// TIA Portal project "Motion_Control" (V17)

(* hardware
DEVICE "HMI_1"  KTP700 Basic PN
   slot 0: "HMI_1"  KTP700 Basic PN  6AV2 123-2GB03-0AX0  17.0.0.0
   slot 1: "HMI_RT_1"  KTP700 Basic PN  6AV2 123-2GB03-0AX0  17.0.0.0
   slot 5: "HMI_1.IE_CP_1"  PROFINET Interface  17.0.0.0
      slot 1: "PROFINET Interface_1"  PROFINET Interface
         slot 1: "Port_1"  Port
DEVICE "S7-1200 station_1"  S7-1200 Station
   slot 0: "Rack_0"  S7-1200 Rack  Rack  V1.0
   slot 1: "PLC_2"  CPU 1212C DC/DC/DC  6ES7 212-1AE40-0XB0  V4.5
*)

// ===== PLC "PLC_2"  CPU 1212C DC/DC/DC =====

VAR_GLOBAL   // PLC tag table "Default tag table"
   "Axis_1_Pulse" AT %Q0.0 : Bool;
   "Axis_1_Direction" AT %Q0.1 : Bool;
   "Axis_1_Homing switch" AT %I0.0 : Bool;
   "Axis_1_LowHwLimitSwitch" AT %I0.1 : Bool;
   "Axis_1_HighHwLimitSwitch" AT %I0.2 : Bool;
   "HMI Driver Start Stop" AT %M10.0 : Bool;
   "Axis 1 Driver Disable" AT %Q0.2 : Bool;
   "Error Power" AT %MW20 : Word;
   "HMI Home Position" AT %M10.1 : Bool;
   "Error Homing" AT %MW22 : Word;
   "HMI CCW" AT %M10.2 : Bool;
   "HMI CW" AT %M10.3 : Bool;
   "Error MoveJog" AT %MW24 : Word;
   "HMI Relative Button" AT %M10.4 : Bool;
   "Error Relative" AT %MW26 : Word;
   "HMI Distance Input" AT %MD28 : Real;
   "Real Distance Input" AT %MD32 : Real;
   "HMI Absolute Button" AT %M10.5 : Bool;
   "Error Absolute" AT %MW36 : Word;
   "HMI Stop Button" AT %M10.6 : Bool;
   "Error Halt" AT %MW38 : Word;
   "HMI System Reset" AT %M10.7 : Bool;
   "Error Reset" AT %MW40 : Word;
   "Position Memory" AT %MD42 : Real;
   "Position Value" AT %MD46 : Real;
   "Velocity Value" AT %MD50 : Real;
   "Velocity Go" AT %M11.0 : Bool;
   "HMI Movement 1" AT %M11.1 : Bool;
   "Tag_1" AT %M11.2 : Bool;
   "Error CT" AT %MW54 : Word;
END_VAR

// folder: System blocks/Program resources

DATA_BLOCK "Timer System Stop"   // DB9
{ S7_Optimized_Access := 'TRUE' }
AUTHOR : Simatic
FAMILY : IEC
NAME : IEC_TMR
VERSION : 1.0
// stored: InstanceOfName IEC_TIMER
"IEC_TIMER"
BEGIN
END_DATA_BLOCK

// folder: (top level)

DATA_BLOCK "Axis_1"   // DB1, Motion_DB
{ S7_Optimized_Access := 'TRUE' }
AUTHOR : SIMATIC
FAMILY : BasicMC
NAME : TO_PosAx
VERSION : 7.0
// stored: InstanceOfName TO_PositioningAxis
"TO_PositioningAxis"
BEGIN
   // Axis.PositionLimitsMax_AddressCU = %I0.2
   // Axis.PositionLimitsMin_AddressCU = %I0.1
   // Axis.PassiveHomingReferencePointSwitch_AddressCU = %I0.0
   // Axis.HomingReferencePointSwitch_AddressCU = %I0.0
   // Axis.NormalizedMaxVelocity.Input = 360.0
   // Axis.LengthUnitNormalized.Distance = 1005
   // Axis.OnlinePtoModeCU = 16#0000_0002
   // Axis.DirectionOutputEnabledCU = TRUE
   // Axis.SelectedChannel2EnumCU = %Q0.1
   // Axis.SelectedChannel1EnumCU = %Q0.0
   // Pulse.MinDeltaDeltaFrequencyCU = 0.004
   // Pulse.MaxDeltaDeltaFrequencyCU = 1.0E+10
   // Pulse.MinDeltaFrequencyCU = 0.005
   // Pulse.MaxDeltaFrequencyCU = 9.5E+9
   // Pulse.MinFrequencyCU = 1.0
   // Pulse.MaxFrequencyCU = 100000.0
   // Pulse.OutputSourceCU = 16#0000_0000
   // Axis.SelectPTO = 0
   // Axis.LengthUnit.LastDistance = 1005
END_DATA_BLOCK

DATA_BLOCK "Movement Table"   // DB10, BMC_202
{ S7_Optimized_Access := 'TRUE' }
AUTHOR : SIMATIC
FAMILY : BasicMC
NAME : CmdTab
VERSION : 7.0
// stored: InstanceOfName TO_CommandTable
"TO_CommandTable"
BEGIN
   // BasicMotionControl.CompileUnit.ExtendedGeneral.ConnectedAxisDBName = Axis_1
   // BasicMotionControl.CompileUnit.ExtendedGeneral.UsedParameters = 1
   // BasicMotionControl.CompileUnit.ExtendedGeneral.AxisID = {2232340-4704}
END_DATA_BLOCK

ORGANIZATION_BLOCK "Main"   // OB1, LAD, ProgramCycle
TITLE = "Main Program Sweep (Cycle)"
{ S7_Optimized_Access := 'TRUE' }
VERSION : 0.1
   VAR_INPUT
      Initial_Call : Bool;   // Initial call of this OB
      Remanence : Bool;   // =True, if remanent data are available
   END_VAR
   VAR_TEMP   // added for the SCL form of the ladder/FBD networks
      _w1 : Bool;
   END_VAR
BEGIN

REGION Network 1: Commissioning the driver
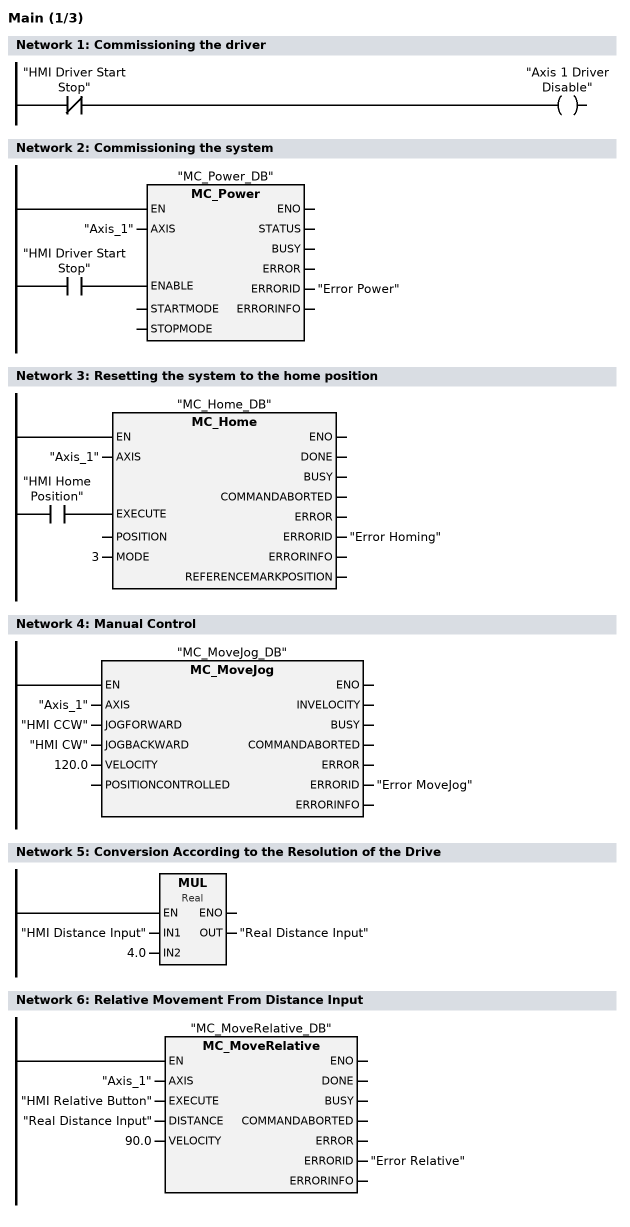
   RUNG wire#powerrail
      I_Contact( "HMI Driver Start Stop" )
      Coil( "Axis 1 Driver Disable" )
   END_RUNG
   // the same network as SCL:
   "Axis 1 Driver Disable" := NOT "HMI Driver Start Stop";
END_REGION

REGION Network 2: Commissioning the system
   "MC_Power_DB"(Axis := "Axis_1", Enable := "HMI Driver Start Stop", ErrorID => "Error Power");   // MC_Power
END_REGION

REGION Network 3: Resetting the system to the home position
   "MC_Home_DB"(Axis := "Axis_1", Execute := "HMI Home Position", Mode := 3, ErrorID => "Error Homing");   // MC_Home
END_REGION

REGION Network 4: Manual Control
   "MC_MoveJog_DB"(Axis := "Axis_1",   // MC_MoveJog
                   JogForward := "HMI CCW",
                   JogBackward := "HMI CW",
                   Velocity := 120.0,
                   ErrorID => "Error MoveJog");
END_REGION

REGION Network 5: Conversion According to the Resolution of the Drive
   RUNG wire#powerrail
      { S7_Templates := "SrcType := Real" } Mul(in1 := "HMI Distance Input", in2 := 4.0, out => "Real Distance Input")
   END_RUNG
   // the same network as SCL:
   "Real Distance Input" := "HMI Distance Input" * 4.0;
END_REGION

REGION Network 6: Relative Movement From Distance Input
   "MC_MoveRelative_DB"(Axis := "Axis_1",   // MC_MoveRelative
                        Execute := "HMI Relative Button",
                        Distance := "Real Distance Input",
                        Velocity := 90.0,
                        ErrorID => "Error Relative");
END_REGION

REGION Network 7: Absolute Movement From Distance Input
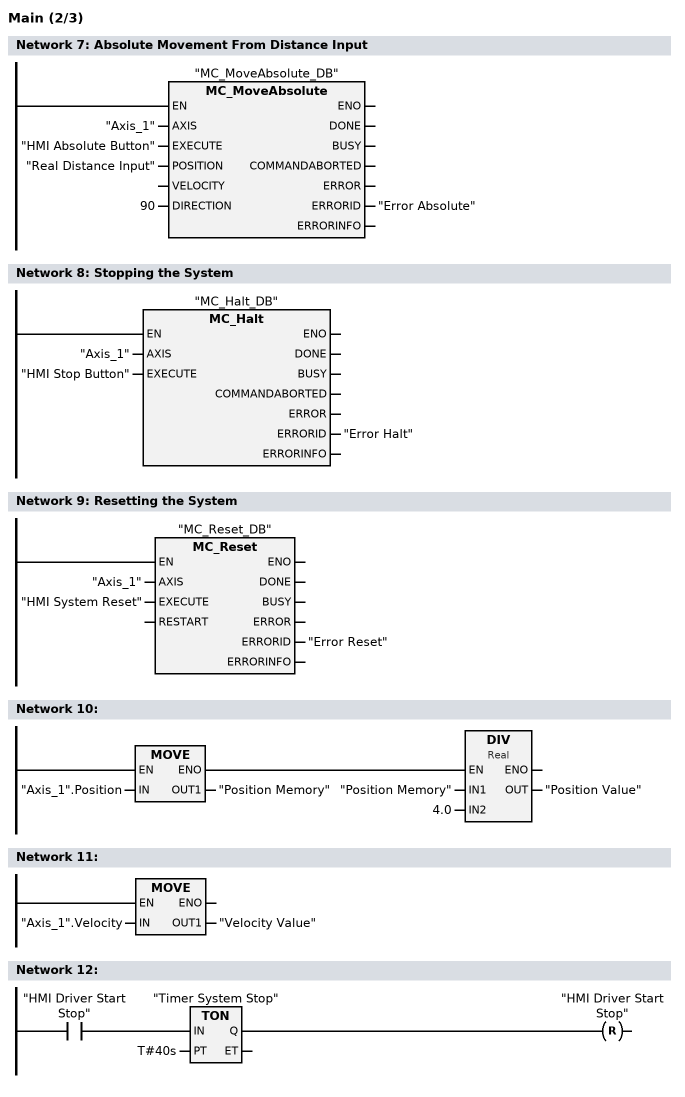
   "MC_MoveAbsolute_DB"(Axis := "Axis_1",   // MC_MoveAbsolute
                        Execute := "HMI Absolute Button",
                        Position := "Real Distance Input",
                        Direction := 90,
                        ErrorID => "Error Absolute");
END_REGION

REGION Network 8: Stopping the System
   "MC_Halt_DB"(Axis := "Axis_1", Execute := "HMI Stop Button", ErrorID => "Error Halt");   // MC_Halt
END_REGION

REGION Network 9: Resetting the System
   "MC_Reset_DB"(Axis := "Axis_1", Execute := "HMI System Reset", ErrorID => "Error Reset");   // MC_Reset
END_REGION

REGION Network 10
   RUNG wire#powerrail
      Move(in := "Axis_1".Position, out1 => "Position Memory")
      { S7_Templates := "SrcType := Real" } Div(in1 := "Position Memory", in2 := 4.0, out => "Position Value")
   END_RUNG
   // the same network as SCL:
   "Position Memory" := "Axis_1".Position;
   "Position Value" := "Position Memory" / 4.0;
END_REGION

REGION Network 11
   RUNG wire#powerrail
      Move(in := "Axis_1".Velocity, out1 => "Velocity Value")
   END_RUNG
   // the same network as SCL:
   "Velocity Value" := "Axis_1".Velocity;
END_REGION

REGION Network 12
   "Timer System Stop".TON(IN := "HMI Driver Start Stop", PT := T#40s);
   IF "Timer System Stop".Q THEN "HMI Driver Start Stop" := FALSE; END_IF;
END_REGION

REGION Network 13
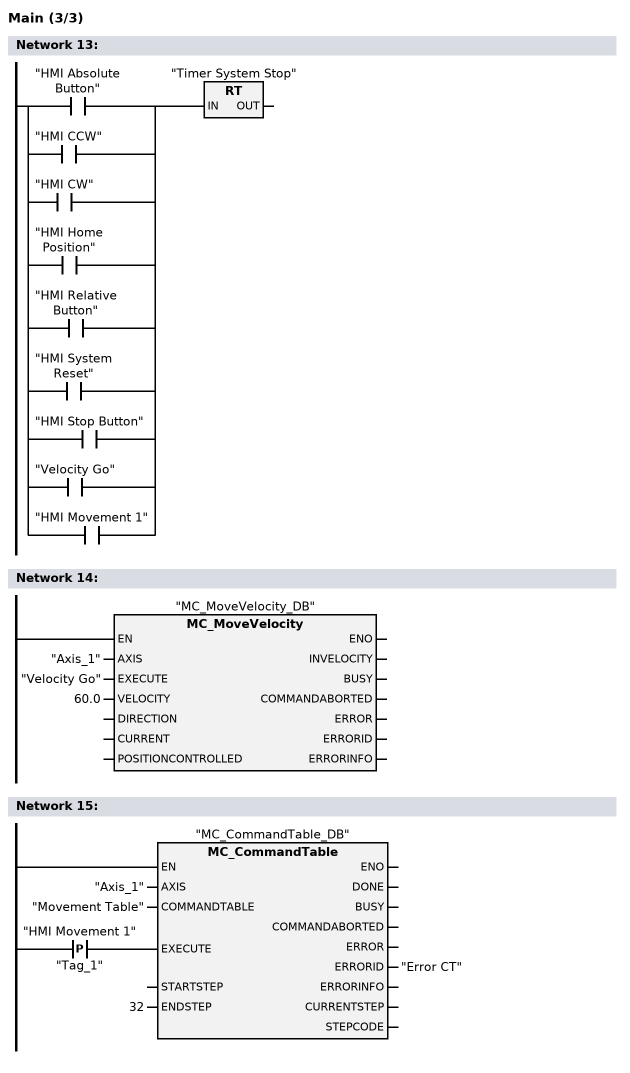
   RUNG wire#powerrail
      Contact( "HMI Absolute Button" )
      wire#w1
      RT_Coil( "Timer System Stop" )
   END_RUNG
   RUNG wire#powerrail
      Contact( "HMI CCW" )
   END_RUNG wire#w1
   RUNG wire#powerrail
      Contact( "HMI CW" )
   END_RUNG wire#w1
   RUNG wire#powerrail
      Contact( "HMI Home Position" )
   END_RUNG wire#w1
   RUNG wire#powerrail
      Contact( "HMI Relative Button" )
   END_RUNG wire#w1
   RUNG wire#powerrail
      Contact( "HMI System Reset" )
   END_RUNG wire#w1
   RUNG wire#powerrail
      Contact( "HMI Stop Button" )
   END_RUNG wire#w1
   RUNG wire#powerrail
      Contact( "Velocity Go" )
   END_RUNG wire#w1
   RUNG wire#powerrail
      Contact( "HMI Movement 1" )
   END_RUNG wire#w1
   // the same network as SCL:
   IF "HMI Absolute Button" OR "HMI CCW" OR "HMI CW" OR "HMI Home Position" OR "HMI Relative Button" OR "HMI System Reset" OR "HMI Stop Button" OR "Velocity Go" OR "HMI Movement 1" THEN
       RESET_TIMER("Timer System Stop");
   END_IF;
END_REGION

REGION Network 14
   "MC_MoveVelocity_DB"(Axis := "Axis_1", Execute := "Velocity Go", Velocity := 60.0);   // MC_MoveVelocity
END_REGION

REGION Network 15
   #_w1 := "HMI Movement 1" AND NOT "Tag_1";   // rising edge of "HMI Movement 1"
   "Tag_1" := "HMI Movement 1";
   "MC_CommandTable_DB"(Axis := "Axis_1",   // MC_CommandTable
                        CommandTable := "Movement Table",
                        Execute := #_w1,
                        EndStep := 32,
                        ErrorID => "Error CT");
END_REGION
END_ORGANIZATION_BLOCK

(* ===== HMI "HMI_RT_1" =====
system functions are stored by id; their names below are inferred from use
connection "HMI_Connection_1": ETHERNET, SMART_S7_1200_OMS

HMI tags "Default tag table"
   "sdfsdf" : Bool = PLC sdfsdf AT %M0.0, 1 s
   "HMI Driver Start Stop" : Bool = PLC "HMI Driver Start Stop" AT %M10.0, 1 s
   "HMI CW" : Bool = PLC "HMI CW" AT %M10.3, 1 s
   "HMI CCW" : Bool = PLC "HMI CCW" AT %M10.2, 1 s
   "HMI Home Position" : Bool = PLC "HMI Home Position" AT %M10.1, 1 s
   "HMI Stop Button" : Bool = PLC "HMI Stop Button" AT %M10.6, 1 s
   "HMI System Reset" : Bool = PLC "HMI System Reset" AT %M10.7, 1 s
   "HMI Absolute Button" : Bool = PLC "HMI Absolute Button" AT %M10.5, 1 s
   "HMI Relative Button" : Bool = PLC "HMI Relative Button" AT %M10.4, 1 s
   "Axis 1 Driver Disable" : Bool = PLC "Axis 1 Driver Disable" AT %Q0.2, 1 s
   "Position Value" : Real = PLC "Position Value" AT %MD46, 1 s
   "Velocity Value" : Real = PLC "Velocity Value" AT %MD50, 1 s
   "HMI Distance Input" : Real = PLC "HMI Distance Input" AT %MD28, 1 s
   "HMI Movement 1" : Bool = PLC "HMI Movement 1" AT %M11.1, 1 s

Template "Template_1" 800x480
   Softkey "Softkey_F1" at 0,0 size 0x0
      on KeyDown: ActivateScreen("Manual", 0)

screen "Manual" 800x480, template "Template_1"
   TextField "Text field_1" at 261,7 size 278x27; Text 'MANUAL MOTION CONTROL'
   Button "Button_1" at 66,74 size 150x75; TextOff 'SYSTEM START/STOP'
      on Press: InvertBit("HMI Driver Start Stop")
   Circle "Circle_1" at 321,97 size 35x35
      Appearance <- "Axis 1 Driver Disable"
   Button "Button_2" at 64,173 size 75x45; TextOff 'CCW'
      on Release: ResetBit("HMI CCW")
      on Press: SetBit("HMI CCW")
   Button "Button_3" at 143,173 size 75x45; TextOff 'CW'
      on Press: SetBit("HMI CW")
      on Release: ResetBit("HMI CW")
   IOField "I/O field_1" at 469,98 size 74x34; FormatPattern s9999
      ProcessValue <- "Position Value"
   TextField "Text field_2" at 459,73 size 92x25; Text 'POSITION'
   IOField "I/O field_2" at 651,98 size 74x34; FormatPattern 9999
      ProcessValue <- "Velocity Value"
   TextField "Text field_3" at 658,73 size 58x23; Text 'SPEED'
   Button "Button_4" at 322,173 size 402x45; TextOff 'REVERT HOME POSITION'
      on Press: SetBit("HMI Home Position")
      on Release: ResetBit("HMI Home Position")
   Button "Button_5" at 104,230 size 75x45; TextOff 'STOP'
      on Release: ResetBit("HMI Stop Button")
      on Press: SetBit("HMI Stop Button")
   Button "Button_6" at 321,297 size 184x45; TextOff 'ABSOLUTE MOVEMENT'
      on Release: ResetBit("HMI Absolute Button")
      on Press: SetBit("HMI Absolute Button")
   Button "Button_7" at 321,361 size 184x45; TextOff 'RELATIVE MOVEMENT'
      on Press: SetBit("HMI Relative Button")
      on Release: ResetBit("HMI Relative Button")
   IOField "I/O field_3" at 586,347 size 74x34; FormatPattern s9999
      ProcessValue <- "HMI Distance Input"
   TextField "Text field_4" at 583,319 size 135x25; Text 'Enter Distance:'
   Button "Button_8" at 67,318 size 150x75; TextOff 'SYSTEM RESET'
      on Press: SetBit("HMI System Reset")
      on Release: ResetBit("HMI System Reset")
   TextField "Text field_5" at 724,434 size 49x23; Text 'NEXT'
   TextField "Text field_6" at 724,451 size 50x23; Text 'PAGE'
   Softkey "Softkey_F8" at 0,0 size 0x0
      on KeyDown: ActivateScreen("Automatic", 0)

screen "Automatic" 800x480, template "Template_1"
   TextField "Text field_1" at 253,7 size 313x27; Text 'AUTOMATIC MOTION CONTROL'
   TextField "Text field_2" at 603,434 size 90x23; Text 'PREVIOUS'
   TextField "Text field_3" at 620,451 size 50x23; Text 'PAGE'
   TextField "Text field_4" at 22,435 size 50x23; Text 'MAIN'
   TextField "Text field_5" at 22,452 size 50x23; Text 'PAGE'
   IOField "I/O field_1" at 469,98 size 74x34; FormatPattern s9999
      ProcessValue <- "Position Value"
   TextField "Text field_6" at 459,73 size 92x25; Text 'POSITION'
   IOField "I/O field_2" at 651,98 size 74x34; FormatPattern 9999
      ProcessValue <- "Velocity Value"
   TextField "Text field_7" at 658,73 size 58x23; Text 'SPEED'
   Button "Button_4" at 33,86 size 402x45; TextOff 'REVERT HOME POSITION'
      on Release: ResetBit("HMI Home Position")
      on Press: SetBit("HMI Home Position")
   Button "Button_1" at 33,161 size 692x49; TextOff 'RUN ACCORDING TO THE MOVEMENT TABLE'
      on Press: SetBit("HMI Movement 1")
      on Release: ResetBit("HMI Movement 1")
   Softkey "Softkey_F7" at 0,0 size 0x0
      on KeyDown: ActivateScreen("Manual", 0)
*)